SUBAPPLICATION Speedcalculation (* Subapplication Type *)
  (* Standard: 61499-2 *)
  (* Version 1.0, 2026-03-23, 04jul *)
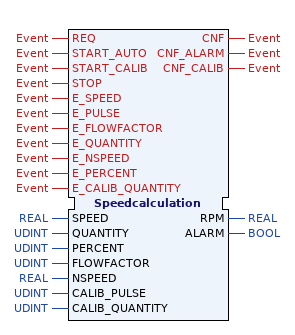
  EVENT_INPUT
    REQ;
    START_AUTO;
    START_CALIB;
    STOP;
    E_SPEED;
    E_PULSE;
    E_FLOWFACTOR;
    E_QUANTITY;
    E_NSPEED;
    E_PERCENT;
    E_CALIB_QUANTITY;
  END_EVENT
  EVENT_OUTPUT
    CNF;
    CNF_ALARM;
    CNF_CALIB;
  END_EVENT
  VAR_INPUT
    SPEED : REAL;
    QUANTITY : UDINT;
    PERCENT : UDINT;
    FLOWFACTOR : UDINT;
    NSPEED : REAL;
    CALIB_PULSE : UDINT;
    CALIB_QUANTITY : UDINT;
  END_VAR
  VAR_OUTPUT
    RPM : REAL;
    ALARM : BOOL;
  END_VAR
  FBS
    F_DIV : iec61131::arithmetic::F_DIV(IN2 := REAL#3.6);
    F_DIV_1 : iec61131::arithmetic::F_DIV;
    F_UDINT_TO_REAL : iec61131::conversion::F_UDINT_TO_REAL;
    F_UDINT_TO_REAL_1 : iec61131::conversion::F_UDINT_TO_REAL;
    F_MUL : iec61131::arithmetic::F_MUL(IN2 := UDINT#12);
    F_REAL_TO_UDINT : iec61131::conversion::F_REAL_TO_UDINT;
    F_EQ : iec61131::comparison::F_GE;
    F_UDINT_TO_REAL_2 : iec61131::conversion::F_UDINT_TO_REAL;
    F_LREAL_TO_UDINT : iec61131::conversion::F_REAL_TO_UDINT;
    SEL_SPEED : iec61131::selection::F_SEL(IN0 := REAL#0.0);
    F_MOVE : iec61131::selection::F_MOVE;
    F_SUB : iec61131::arithmetic::F_SUB;
    F_UDINT_TO_REAL_3 : iec61131::conversion::F_UDINT_TO_REAL;
    F_UDINT_TO_REAL_4 : iec61131::conversion::F_UDINT_TO_REAL;
    F_REAL_TO_UDINT_1 : iec61131::conversion::F_REAL_TO_UDINT;
    m2_s : iec61131::arithmetic::F_MUL(IN2 := LREAL#3.5);
    F_REAL_TO_LREAL : iec61131::conversion::F_REAL_TO_LREAL;
    g_s : iec61131::arithmetic::F_MUL;
    F_LREAL_TO_REAL : iec61131::conversion::F_LREAL_TO_REAL;
    F_DIV_2 : iec61131::arithmetic::F_DIV(IN2 := LREAL#10000.0);
    F_UDINT_TO_REAL_5 : iec61131::conversion::F_UDINT_TO_LREAL;
    F_LREAL_TO_REAL_1 : iec61131::conversion::F_LREAL_TO_REAL;
    g_min : iec61131::arithmetic::F_MUL(IN2 := LREAL#60.0);
    F_REAL_TO_LREAL_1 : iec61131::conversion::F_REAL_TO_LREAL;
    F_UDINT_TO_REAL_6 : iec61131::conversion::F_UDINT_TO_REAL;
    F_LREAL_TO_UDINT_1 : iec61131::conversion::F_LREAL_TO_REAL;
    u_min : iec61131::arithmetic::F_DIV;
    F_REAL_TO_LREAL_2 : iec61131::conversion::F_REAL_TO_LREAL;
    F_GE : iec61131::comparison::F_GE(IN2 := LREAL#55.0);
    F_SEL_E_3 : eclipse4diac::utils::selection::F_SEL_E_3(IN1 := REAL#0.0);
    F_REAL_TO_LREAL_3 : iec61131::conversion::F_REAL_TO_LREAL;
    F_UDINT_TO_REAL_7 : iec61131::conversion::F_UDINT_TO_LREAL;
    F_DIV_3 : iec61131::arithmetic::F_DIV(IN2 := REAL#3.6);
    F_DIV_4 : iec61131::arithmetic::F_DIV(IN2 := LREAL#10000.0);
    F_REAL_TO_LREAL_4 : iec61131::conversion::F_REAL_TO_LREAL;
    m2_s_1 : iec61131::arithmetic::F_MUL(IN2 := LREAL#3.5);
    F_LREAL_TO_REAL_3 : iec61131::conversion::F_LREAL_TO_REAL;
    F_LREAL_TO_REAL_4 : iec61131::conversion::F_LREAL_TO_REAL;
    g_s_1 : iec61131::arithmetic::F_MUL;
    F_REAL_TO_LREAL_5 : iec61131::conversion::F_REAL_TO_LREAL;
    g_min_1 : iec61131::arithmetic::F_MUL(IN2 := LREAL#60.0);
    F_LREAL_TO_UDINT_2 : iec61131::conversion::F_LREAL_TO_REAL;
    F_UDINT_TO_REAL_8 : iec61131::conversion::F_UDINT_TO_REAL;
    u_min_1 : iec61131::arithmetic::F_DIV;
    F_REAL_TO_LREAL_6 : iec61131::conversion::F_REAL_TO_LREAL;
    E_PERMIT : iec61499::events::E_PERMIT;
    AUTO : iec61499::events::E_RS;
    CALIB : iec61499::events::E_RS;
    E_PERMIT_1 : iec61499::events::E_PERMIT;
    E_PERMIT_2 : iec61499::events::E_PERMIT;
    E_PERMIT_3 : iec61499::events::E_PERMIT;
    E_PERMIT_4 : iec61499::events::E_PERMIT;
  END_FBS
  EVENT_CONNECTIONS
    E_NSPEED TO F_DIV.REQ;
    F_UDINT_TO_REAL.CNF TO F_DIV_1.REQ;
    E_CALIB_QUANTITY TO F_UDINT_TO_REAL.REQ;
    F_UDINT_TO_REAL_1.CNF TO F_DIV_1.REQ;
    E_FLOWFACTOR TO F_UDINT_TO_REAL_1.REQ;
    F_DIV_1.CNF TO F_REAL_TO_UDINT.REQ;
    F_REAL_TO_UDINT.CNF TO F_MUL.REQ;
    F_UDINT_TO_REAL_2.CNF TO F_LREAL_TO_UDINT.REQ;
    F_MUL.CNF TO F_UDINT_TO_REAL_2.REQ;
    F_LREAL_TO_UDINT.CNF TO F_EQ.REQ;
    F_EQ.CNF TO SEL_SPEED.REQ;
    START_CALIB TO F_MOVE.REQ;
    F_MOVE.CNF TO F_UDINT_TO_REAL_3.REQ;
    F_UDINT_TO_REAL_3.CNF TO F_SUB.REQ;
    F_UDINT_TO_REAL_4.CNF TO F_SUB.REQ;
    E_PULSE TO E_PERMIT_2.EI;
    F_REAL_TO_UDINT_1.CNF TO F_EQ.REQ;
    F_SUB.CNF TO F_REAL_TO_UDINT_1.REQ;
    F_DIV.CNF TO F_REAL_TO_LREAL.REQ;
    F_REAL_TO_LREAL.CNF TO m2_s.REQ;
    m2_s.CNF TO F_LREAL_TO_REAL.REQ;
    F_LREAL_TO_REAL.CNF TO g_s.REQ;
    F_UDINT_TO_REAL_5.CNF TO F_DIV_2.REQ;
    E_QUANTITY TO F_UDINT_TO_REAL_5.REQ;
    F_DIV_2.CNF TO F_LREAL_TO_REAL_1.REQ;
    F_LREAL_TO_REAL_1.CNF TO g_s.REQ;
    g_s.CNF TO F_REAL_TO_LREAL_1.REQ;
    F_REAL_TO_LREAL_1.CNF TO g_min.REQ;
    g_min.CNF TO F_LREAL_TO_UDINT_1.REQ;
    E_FLOWFACTOR TO F_UDINT_TO_REAL_6.REQ;
    F_LREAL_TO_UDINT_1.CNF TO u_min.REQ;
    F_UDINT_TO_REAL_6.CNF TO u_min.REQ;
    u_min.CNF TO F_REAL_TO_LREAL_2.REQ;
    F_REAL_TO_LREAL_2.CNF TO F_GE.REQ;
    F_GE.CNF TO CNF_ALARM;
    F_SEL_E_3.CNF TO CNF;
    SEL_SPEED.CNF TO F_REAL_TO_LREAL_3.REQ;
    F_REAL_TO_LREAL_3.CNF TO E_PERMIT_3.EI;
    STOP TO F_SEL_E_3.REQ1;
    F_LREAL_TO_REAL_3.CNF TO g_s_1.REQ;
    F_DIV_3.CNF TO F_REAL_TO_LREAL_4.REQ;
    E_FLOWFACTOR TO F_UDINT_TO_REAL_8.REQ;
    m2_s_1.CNF TO F_LREAL_TO_REAL_3.REQ;
    F_UDINT_TO_REAL_7.CNF TO F_DIV_4.REQ;
    F_REAL_TO_LREAL_4.CNF TO m2_s_1.REQ;
    g_min_1.CNF TO F_LREAL_TO_UDINT_2.REQ;
    F_LREAL_TO_UDINT_2.CNF TO u_min_1.REQ;
    E_QUANTITY TO F_UDINT_TO_REAL_7.REQ;
    g_s_1.CNF TO F_REAL_TO_LREAL_5.REQ;
    F_UDINT_TO_REAL_8.CNF TO u_min_1.REQ;
    F_LREAL_TO_REAL_4.CNF TO g_s_1.REQ;
    F_DIV_4.CNF TO F_LREAL_TO_REAL_4.REQ;
    F_REAL_TO_LREAL_5.CNF TO g_min_1.REQ;
    E_SPEED TO E_PERMIT.EI;
    F_REAL_TO_LREAL_2.CNF TO SEL_SPEED.REQ;
    u_min_1.CNF TO F_REAL_TO_LREAL_6.REQ;
    F_REAL_TO_LREAL_6.CNF TO E_PERMIT_4.EI;
    E_PERMIT.EO TO F_DIV_3.REQ;
    START_AUTO TO AUTO.S;
    STOP TO AUTO.R;
    STOP TO CALIB.R;
    START_CALIB TO CALIB.S;
    CALIB.EO TO E_PERMIT_1.EI;
    E_PERMIT_1.EO TO F_MOVE.REQ;
    E_PERMIT_2.EO TO F_UDINT_TO_REAL_4.REQ;
    E_PERMIT_3.EO TO F_SEL_E_3.REQ3;
    E_PERMIT_4.EO TO F_SEL_E_3.REQ2;
  END_CONNECTIONS
  DATA_CONNECTIONS
    NSPEED TO F_DIV.IN1;
    CALIB_QUANTITY TO F_UDINT_TO_REAL.IN;
    F_UDINT_TO_REAL.OUT TO F_DIV_1.IN1;
    F_UDINT_TO_REAL_1.OUT TO F_DIV_1.IN2;
    FLOWFACTOR TO F_UDINT_TO_REAL_1.IN;
    F_DIV_1.OUT TO F_REAL_TO_UDINT.IN;
    F_REAL_TO_UDINT.OUT TO F_MUL.IN1;
    F_UDINT_TO_REAL_2.OUT TO F_LREAL_TO_UDINT.IN;
    F_MUL.OUT TO F_UDINT_TO_REAL_2.IN;
    F_LREAL_TO_UDINT.OUT TO F_EQ.IN1;
    F_EQ.OUT TO SEL_SPEED.G;
    CALIB_PULSE TO F_MOVE.IN;
    F_MOVE.OUT TO F_UDINT_TO_REAL_3.IN;
    F_UDINT_TO_REAL_3.OUT TO F_SUB.IN2;
    F_UDINT_TO_REAL_4.OUT TO F_SUB.IN1;
    CALIB_PULSE TO F_UDINT_TO_REAL_4.IN;
    F_SUB.OUT TO F_REAL_TO_UDINT_1.IN;
    F_REAL_TO_UDINT_1.OUT TO F_EQ.IN2;
    F_DIV.OUT TO F_REAL_TO_LREAL.IN;
    F_REAL_TO_LREAL.OUT TO m2_s.IN1;
    m2_s.OUT TO F_LREAL_TO_REAL.IN;
    F_LREAL_TO_REAL.OUT TO g_s.IN1;
    F_UDINT_TO_REAL_5.OUT TO F_DIV_2.IN1;
    QUANTITY TO F_UDINT_TO_REAL_5.IN;
    F_DIV_2.OUT TO F_LREAL_TO_REAL_1.IN;
    F_LREAL_TO_REAL_1.OUT TO g_s.IN2;
    g_s.OUT TO F_REAL_TO_LREAL_1.IN;
    F_REAL_TO_LREAL_1.OUT TO g_min.IN1;
    g_min.OUT TO F_LREAL_TO_UDINT_1.IN;
    FLOWFACTOR TO F_UDINT_TO_REAL_6.IN;
    F_LREAL_TO_UDINT_1.OUT TO u_min.IN1;
    F_UDINT_TO_REAL_6.OUT TO u_min.IN2;
    u_min.OUT TO F_REAL_TO_LREAL_2.IN;
    F_REAL_TO_LREAL_2.OUT TO F_GE.IN1;
    F_GE.OUT TO ALARM;
    F_SEL_E_3.OUT TO RPM;
    SEL_SPEED.OUT TO F_REAL_TO_LREAL_3.IN;
    F_REAL_TO_LREAL_3.OUT TO F_SEL_E_3.IN3;
    F_REAL_TO_LREAL_4.OUT TO m2_s_1.IN1;
    F_UDINT_TO_REAL_7.OUT TO F_DIV_4.IN1;
    F_DIV_4.OUT TO F_LREAL_TO_REAL_4.IN;
    FLOWFACTOR TO F_UDINT_TO_REAL_8.IN;
    QUANTITY TO F_UDINT_TO_REAL_7.IN;
    F_LREAL_TO_REAL_3.OUT TO g_s_1.IN1;
    g_s_1.OUT TO F_REAL_TO_LREAL_5.IN;
    F_LREAL_TO_UDINT_2.OUT TO u_min_1.IN1;
    F_UDINT_TO_REAL_8.OUT TO u_min_1.IN2;
    F_LREAL_TO_REAL_4.OUT TO g_s_1.IN2;
    F_DIV_3.OUT TO F_REAL_TO_LREAL_4.IN;
    g_min_1.OUT TO F_LREAL_TO_UDINT_2.IN;
    m2_s_1.OUT TO F_LREAL_TO_REAL_3.IN;
    F_REAL_TO_LREAL_5.OUT TO g_min_1.IN1;
    SPEED TO F_DIV_3.IN1;
    F_REAL_TO_LREAL_2.OUT TO SEL_SPEED.IN1;
    u_min_1.OUT TO F_REAL_TO_LREAL_6.IN;
    F_REAL_TO_LREAL_6.OUT TO F_SEL_E_3.IN2;
    AUTO.Q TO E_PERMIT.PERMIT;
    CALIB.Q TO E_PERMIT_1.PERMIT;
    CALIB.Q TO E_PERMIT_2.PERMIT;
    CALIB.Q TO E_PERMIT_3.PERMIT;
    AUTO.Q TO E_PERMIT_4.PERMIT;
  END_CONNECTIONS
END_SUBAPPLICATION
